(*			
	RafalOS
	Rafał Osajda		12.11.2025		TC 4024.66
	interfejs potrzebny w HMI
*)
INTERFACE ITF_HMIEButton_HMI EXTENDS ITF_BaseComponent_HMI

METHOD PUBLIC GetNameOfButton : WSTRING
VAR_INPUT
END_VAR
END_METHOD

METHOD LinkHMIEButtonData : BOOL
VAR_INPUT
	stData					: REFERENCE TO ST_HMIEButton_HMI_Link;
END_VAR
END_METHOD

END_INTERFACE

(* stored: Version 1.1.0.1
   Itf ITF_HMIEButton_HMI: Id {02f9390e-52b4-0016-1a97-38f0c6617069}
   Method GetNameOfButton: Id {bd82dba9-3352-044f-12b2-76cc17ef9ad5}
   Method LinkHMIEButtonData: Id {deb1c421-36cc-02c1-0aa4-1df324480eb1} *)
